FUNCTION_BLOCK Buffer Implements OpenDichtSchuif
VAR_INPUT
END_VAR
VAR_OUTPUT
END_VAR
VAR
END_VAR

// gebruikt lopendeband

END_FUNCTION_BLOCK

(* stored: Version 1.1.0.1
   POU Buffer: Id {f5a9d24e-3f9b-4256-a349-b204b10fe1cf}, SpecialFunc None *)
